{attribute 'qualified_only'}
VAR_GLOBAL
	HVAL_STATUS:			USINT;
	ERROR_STATUS: 			USINT;
	MAX_TEMP: 				UINT;
	emergency_shutdown: 	BOOL;
	total_voltage: UINT;
END_VAR

(* stored: Version 1.1.0.1
   GVL GVL_PT: Id {c13a7a8c-c8d8-41ce-a220-df2a506caa64} *)
